TYPE ST_AnalogInput :
STRUCT
	stStatus AT %I* : ST_AnalogInputStatus;
	nValue AT %I* : INT;
END_STRUCT
END_TYPE

(* stored: Version 1.1.0.1, ProductVersion 3.1.4024.12
   DUT ST_AnalogInput: Id {e158cc4e-06fa-4baa-8a11-8916d6a01a80} *)
